// TIA Portal V19 export
TYPE "LEXCHANGETRAY_typeConstraintRollerIoSignalManualCommands"
// detectionBeforePalletPositioning: Bool
// positioningPinCylinderHomePositionDetection2: Bool
// cellLiftingCylinderHomePositionDetection2: Bool
// positioningPinCylinderWorkingPositionDetection2: Bool
// trayLiftingCylinderWorkingPositionDetection1: Bool
// cellLiftingCylinderWorkingPositionDetection2: Bool
// cellLiftingCylinderHomePositionDetection1: Bool
// trayEntryDetection: Bool
// trayLiftingCylinderHomePositionDetection1: Bool
// positiveLimitForCellJackingAndTransplanting: Bool
// negativeLimitForCellJackingAndTransplanting: Bool
// cellLiftingCylinderWorkingPositionDetection1: Bool
// positioningPinCylinderHomePositionDetection1: Bool
// positioningPinCylinderWorkingPositionDetection1: Bool
// trayInPlaceDetection: Bool
// originalForCellJackingAndTransplanting: Bool
// palletScrewAntiReverseDetection: Bool
// detectionAfterTrayPositioning: Bool
// trayLiftingCylinderHomePositionDetection2: Bool
// trayLiftingCylinderWorkingPositionDetection2: Bool
// stored: Access Published
   STRUCT
      detectionBeforePalletPositioning : Bool;
      positioningPinCylinderHomePositionDetection2 : Bool;
      cellLiftingCylinderHomePositionDetection2 : Bool;
      positioningPinCylinderWorkingPositionDetection2 : Bool;
      trayLiftingCylinderWorkingPositionDetection1 : Bool;
      cellLiftingCylinderWorkingPositionDetection2 : Bool;
      cellLiftingCylinderHomePositionDetection1 : Bool;
      trayEntryDetection : Bool;
      trayLiftingCylinderHomePositionDetection1 : Bool;
      positiveLimitForCellJackingAndTransplanting : Bool;
      negativeLimitForCellJackingAndTransplanting : Bool;
      cellLiftingCylinderWorkingPositionDetection1 : Bool;
      positioningPinCylinderHomePositionDetection1 : Bool;
      positioningPinCylinderWorkingPositionDetection1 : Bool;
      trayInPlaceDetection : Bool;
      originalForCellJackingAndTransplanting : Bool;
      palletScrewAntiReverseDetection : Bool;
      detectionAfterTrayPositioning : Bool;
      trayLiftingCylinderHomePositionDetection2 : Bool;
      trayLiftingCylinderWorkingPositionDetection2 : Bool;
   END_STRUCT;
END_TYPE
